FUNCTION_BLOCK FB_PowerControlledHeaterThyristor EXTENDS FB_ActuatorContinous
VAR_INPUT
	fPowerTotal : REAL;
	fTemperature : REAL;
END_VAR
VAR
	stTemperatureCheckDefaultParameters : ST_RangeCheckDefaultParameters := (tTaskCycleTime := GlobalVariables.tCtrlCycleTime_MAIN, tCtrlCycleTime := GlobalVariables.tCtrlCycleTime_MAIN, fRestoreDifference := 10);
	Temperature_Check : FB_RangeCheck := (ST_DefaultParameters := stTemperatureCheckDefaultParameters);
	
	//controller
	PID_Controller				: FB_CTRL_PID;
	PID_Controller_Parameters	: ST_CTRL_PID_PARAMS;
	
	fSetPoint_internal 			: REAL; //internal setpoint between 0 and 32767
	bTemperaturePermission		: BOOL;
	
	//I/O Links
	nSetPoint_OUT 		AT %Q* : INT;	
	
END_VAR
VAR_OUTPUT
	bError 						: BOOL;
	
END_VAR

Temperature_Check(fInput := fTemperature,
	fLowerLimit := -99,
	fUpperLimit := 100);
bTemperaturePermission := Temperature_Check.bPermission;
	
MAIN();
LocalControl();

METHOD GetState : BOOL
VAR_INPUT
END_VAR
//local state
bStatusOn := controlState.bStatusOn;
END_METHOD

METHOD LocalControl : BOOL
VAR_INPUT
END_VAR
PID_Controller_Parameters.fKp:=1.8;
PID_Controller_Parameters.tTn:= T#1600MS;
PID_Controller_Parameters.tTv:=T#4MS;
PID_Controller_Parameters.fOutMaxLimit:= 32767;
PID_Controller_Parameters.fOutMinLimit:=  0;
PID_Controller_Parameters.tCtrlCycleTime:= T#5S;
PID_Controller_Parameters.tTaskCycleTime:= T#10MS;
PID_Controller_Parameters.bARWOnIPartOnly:= FALSE; 

PID_Controller(fSetpointValue:=fSetPoint, 
fActualValue:=fPowerTotal, 
fManSyncValue:=0, 
bSync:=FALSE, 
eMode:=2, 
bHold:=FALSE, 
stParams:=PID_Controller_Parameters);

//overwrite internal setpoint, if Temperatur is too high
IF bSetStatusOn AND bTemperaturePermission THEN
	fSetPoint_internal := LREAL_TO_REAL(PID_Controller.fOut);
	bError := FALSE;
ELSE
	fSetPoint_internal := 0;
	bError := TRUE;
END_IF
END_METHOD

METHOD PROTECTED  SetSetPointLimits : BOOL
VAR_INPUT
END_VAR
aSetPointLimits[1] := 0;
aSetPointLimits[2] := 5000;
END_METHOD

METHOD SetState : BOOL
VAR_INPUT
END_VAR
setPointState.fSetPoint := fSetPoint_internal;
setPointState.aSetPointLimits := aSetPointLimits;
setPointState.sSetPointUnit := 'W';

nSetPoint_OUT := REAL_TO_INT(fSetPoint_internal);
END_METHOD

END_FUNCTION_BLOCK

(* stored: Version 1.1.0.1, ProductVersion 3.1.4024.6
   POU FB_PowerControlledHeaterThyristor: Id {1501bede-193a-4fe1-a0ad-e0d67950964c}, SpecialFunc None
   Method GetState: Id {8997a89f-b8c8-45e1-a232-72f1814e8bc2}
   Method LocalControl: Id {190aaaaa-eb4b-4ed1-af2c-e7ad87e77bb5}
   Method SetSetPointLimits: Id {2c43ad12-08cc-44af-8962-9730b1a2d0e8}
   Method SetState: Id {f38d706b-6444-4227-a865-784d78405b17} *)
